Staubli VAL3: GetAsyncAxis.pgx

public program GetAsyncAxis(num x_nType (dimensions=1), string& x_sText (dimensions=1), trsf& x_trAxis (dimensions=1))
  local bool l_bBool
  local num l_nBuff
  local num l_nNum
  local string l_sSBuff
begin
  if x_nType!=20 and x_nType!=9
    return
  endIf

  //把第七，第八轴给提取出来
  while find(l_sSBuff,"/")<0 and l_nNum<len(x_sText)
    l_nNum=l_nNum+1
    l_sSBuff=right(x_sText,l_nNum)
  endWhile

  l_sSBuff=right(x_sText,l_nNum-1)+",0,0,0,0"
  x_sText=left(x_sText,len(x_sText)-l_nNum)

  call FileDir:SplitTrsf(l_sSBuff,"",x_trAxis,l_bBool)














end
